FUNCTION_BLOCK SUBL_6 (* Five-variable Local Group Subscriber *)
  (* Standard: 61499-1; Classification: Communications *)
  (* Version 0.0, 2002-05-22, JHC, Rockwell Automation *)
  (* Compiler header: package fb.rt.net; *)
  (* Compiler Java IBM VisualAge 3.0 *)
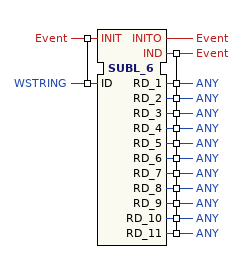
  EVENT_INPUT
    INIT WITH ID; (* Service Initialization *)
  END_EVENT
  EVENT_OUTPUT
    INITO; (* Initialization Confirm *)
    IND WITH RD_1, RD_2, RD_3, RD_4, RD_5, RD_6, RD_7, RD_8, RD_9, RD_10, RD_11; (* Service Indication *)
  END_EVENT
  VAR_INPUT
    ID : WSTRING; (* Local Group Name-Default is FB Instance Name *)
  END_VAR
  VAR_OUTPUT
    RD_1 : ANY; (* Subscribed Data *)
    RD_2 : ANY;
    RD_3 : ANY;
    RD_4 : ANY;
    RD_5 : ANY;
    RD_6 : ANY;
    RD_7 : ANY;
    RD_8 : ANY;
    RD_9 : ANY;
    RD_10 : ANY;
    RD_11 : ANY;
  END_VAR
END_FUNCTION_BLOCK
